// TIA Portal V19 export
FUNCTION "FC_MES" : Void   // FC8, FBD
{ S7_Optimized_Access := 'TRUE' }
// stored: SetENOAutomatically false
BEGIN

REGION Network 1: managen van recipes
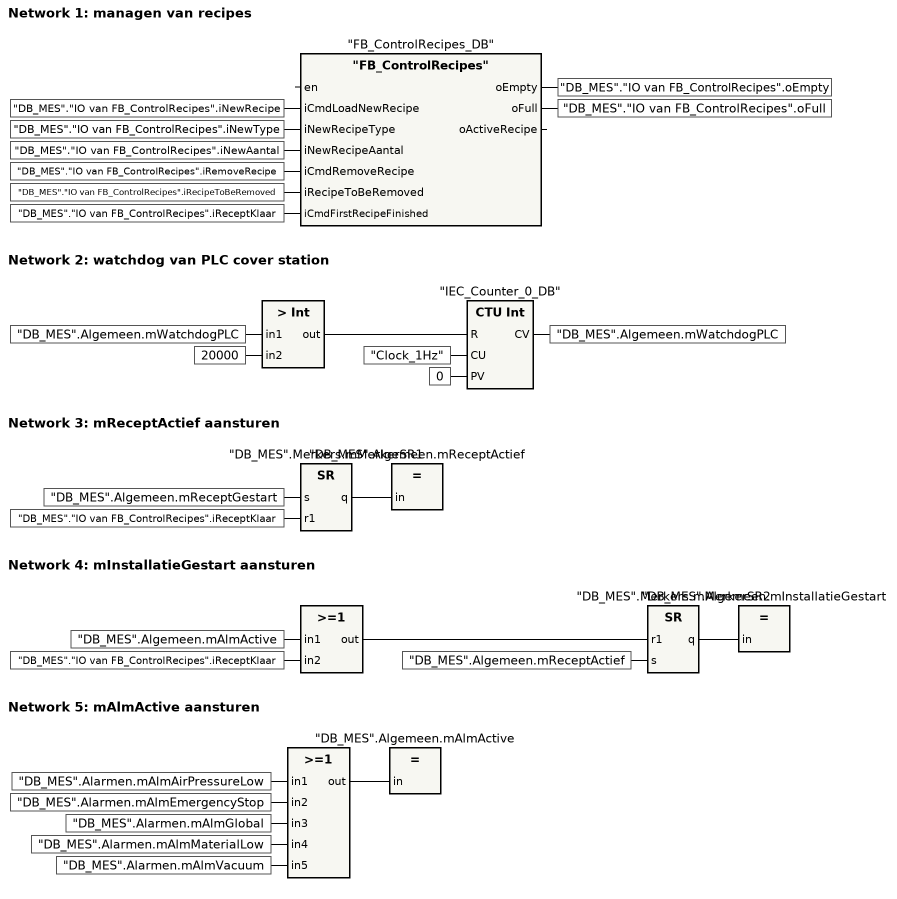
   "FB_ControlRecipes_DB"(iCmdLoadNewRecipe := "DB_MES"."IO van FB_ControlRecipes".iNewRecipe,   // "FB_ControlRecipes"
                          iNewRecipeType := "DB_MES"."IO van FB_ControlRecipes".iNewType,
                          iNewRecipeAantal := "DB_MES"."IO van FB_ControlRecipes".iNewAantal,
                          iCmdRemoveRecipe := "DB_MES"."IO van FB_ControlRecipes".iRemoveRecipe,
                          iRecipeToBeRemoved := "DB_MES"."IO van FB_ControlRecipes".iRecipeToBeRemoved,
                          iCmdFirstRecipeFinished := "DB_MES"."IO van FB_ControlRecipes".iReceptKlaar,
                          oEmpty => "DB_MES"."IO van FB_ControlRecipes".oEmpty,
                          oFull => "DB_MES"."IO van FB_ControlRecipes".oFull);
END_REGION

REGION Network 2: watchdog van PLC cover station
   "IEC_Counter_0_DB".CTU(R := "DB_MES".Algemeen.mWatchdogPLC > 20000,
                          CU := "Clock_1Hz",
                          PV := 0,
                          CV => "DB_MES".Algemeen.mWatchdogPLC);
END_REGION

REGION Network 3: mReceptActief aansturen
   IF "DB_MES".Algemeen.mReceptGestart THEN
       "DB_MES".Merkers.mMerkerSR1 := TRUE;   // SR flip-flop
   END_IF;
   IF "DB_MES"."IO van FB_ControlRecipes".iReceptKlaar THEN "DB_MES".Merkers.mMerkerSR1 := FALSE; END_IF;
   "DB_MES".Algemeen.mReceptActief := "DB_MES".Merkers.mMerkerSR1;
END_REGION

REGION Network 4: mInstallatieGestart aansturen
   IF "DB_MES".Algemeen.mReceptActief THEN
       "DB_MES".Merkers.mMerkerSR2 := TRUE;   // SR flip-flop
   END_IF;
   IF "DB_MES".Algemeen.mAlmActive OR "DB_MES"."IO van FB_ControlRecipes".iReceptKlaar THEN
       "DB_MES".Merkers.mMerkerSR2 := FALSE;
   END_IF;
   "DB_MES".Algemeen.mInstallatieGestart := "DB_MES".Merkers.mMerkerSR2;
END_REGION

REGION Network 5: mAlmActive aansturen
   "DB_MES".Algemeen.mAlmActive := "DB_MES".Alarmen.mAlmAirPressureLow OR "DB_MES".Alarmen.mAlmEmergencyStop OR "DB_MES".Alarmen.mAlmGlobal OR "DB_MES".Alarmen.mAlmMaterialLow OR "DB_MES".Alarmen.mAlmVacuum;
END_REGION

REGION Network 6: schrijven naar node-red
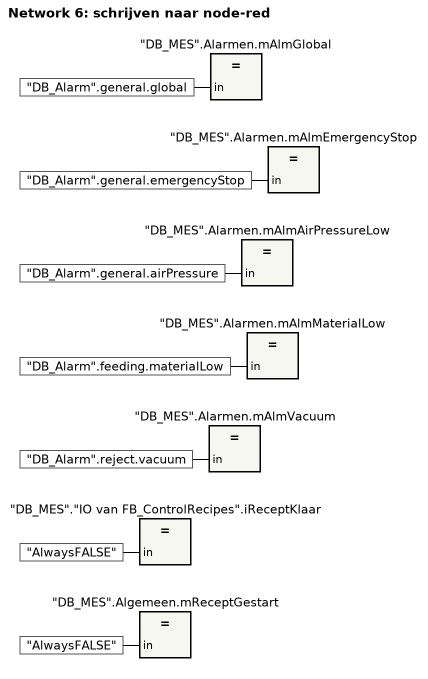
   "DB_MES".Alarmen.mAlmGlobal := "DB_Alarm".general.global;
   "DB_MES".Alarmen.mAlmEmergencyStop := "DB_Alarm".general.emergencyStop;
   "DB_MES".Alarmen.mAlmAirPressureLow := "DB_Alarm".general.airPressure;
   "DB_MES".Alarmen.mAlmMaterialLow := "DB_Alarm".feeding.materialLow;
   "DB_MES".Alarmen.mAlmVacuum := "DB_Alarm".reject.vacuum;
   "DB_MES"."IO van FB_ControlRecipes".iReceptKlaar := "AlwaysFALSE";
   "DB_MES".Algemeen.mReceptGestart := "AlwaysFALSE";
END_REGION
END_FUNCTION
